// SIMATIC S7-200 project (STEP 7-Micro/WIN), CPU 226 REL 02.01

ORGANIZATION_BLOCK Main:OB1
TITLE=程序注释
BEGIN
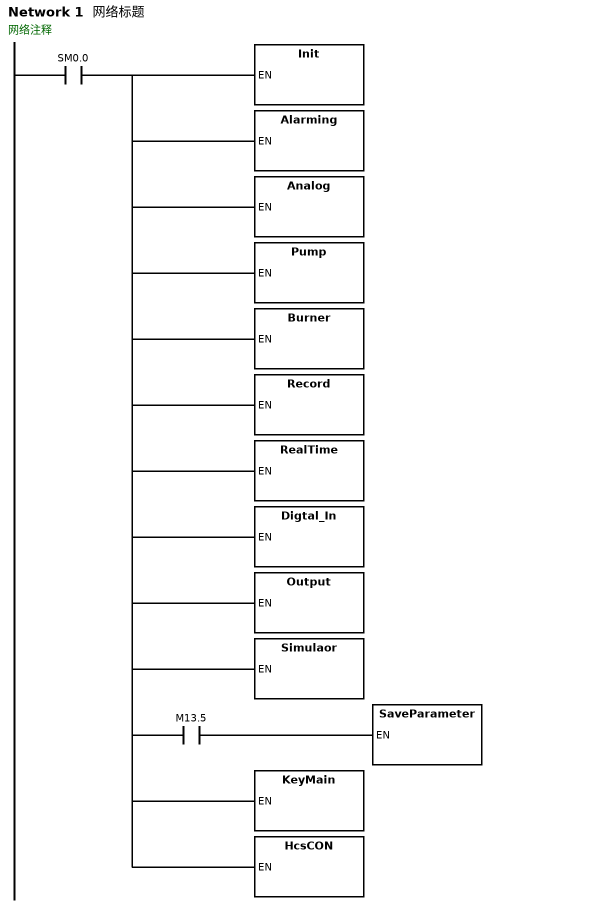
Network 1 // 网络标题
// 网络注释
LD     SM0.0
LPS
CALL   Init:SBR0
CALL   Alarming:SBR4
CALL   Analog:SBR1
CALL   Pump:SBR7
CALL   Burner:SBR14
CALL   Record:SBR11
CALL   RealTime:SBR19
CALL   Digtal_In:SBR17
CALL   Output:SBR24
CALL   Simulaor:SBR25
A      M13.5
CALL   SaveParameter:SBR26
LRD
CALL   KeyMain:SBR28
LPP
CALL   HcsCON:SBR32
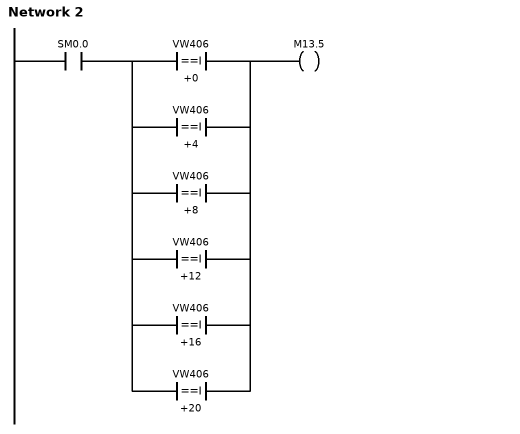
Network 2
LD     SM0.0
LDW=   VW406, +0
OW=    VW406, +4
OW=    VW406, +8
OW=    VW406, +12
OW=    VW406, +16
OW=    VW406, +20
ALD
=      M13.5
END_ORGANIZATION_BLOCK

SUBROUTINE_BLOCK Init:SBR0
TITLE=子程序注释
BEGIN
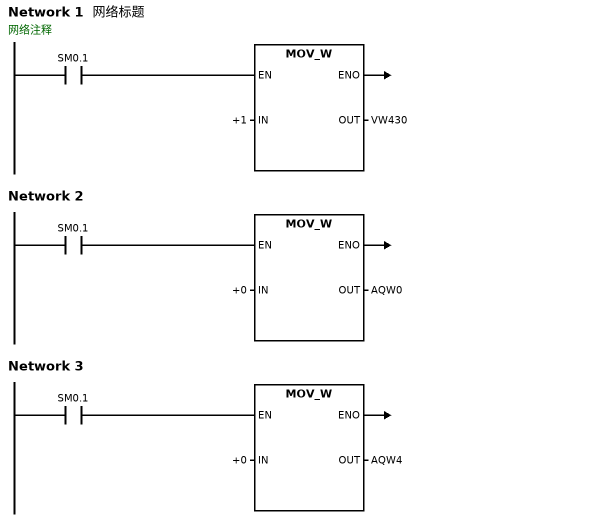
Network 1 // 网络标题
// 网络注释
LD     SM0.1
MOVW   +1, VW430
Network 2
LD     SM0.1
MOVW   +0, AQW0
Network 3
LD     SM0.1
MOVW   +0, AQW4
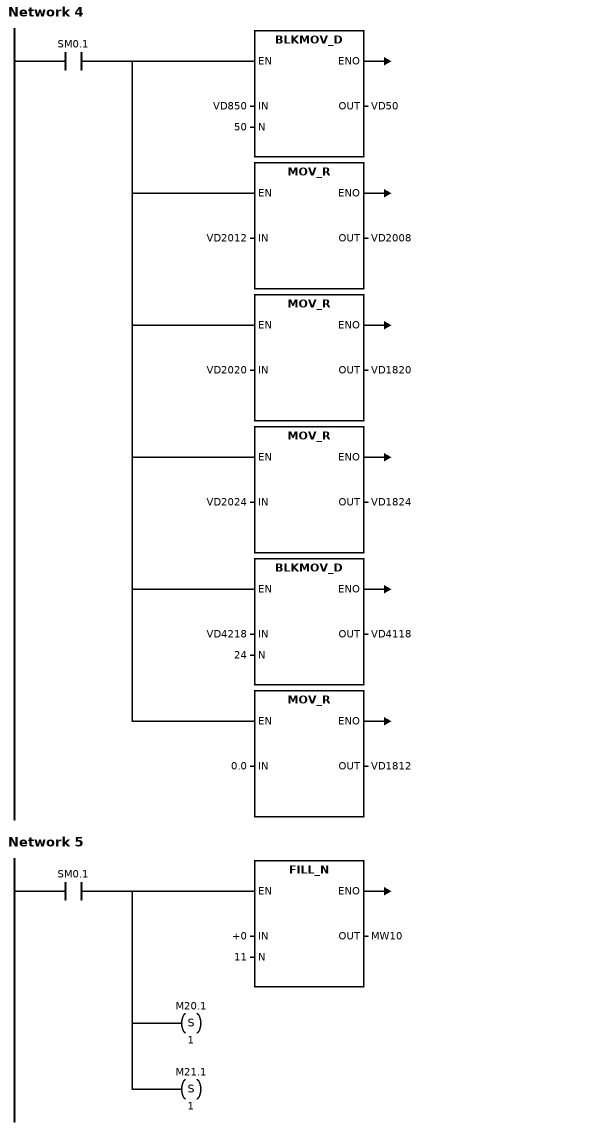
Network 4
LD     SM0.1
BMD    VD850, VD50, 50
MOVR   VD2012, VD2008
MOVR   VD2020, VD1820
MOVR   VD2024, VD1824
BMD    VD4218, VD4118, 24
MOVR   0.0, VD1812
Network 5
LD     SM0.1
FILL   +0, MW10, 11
S      M20.1, 1
S      M21.1, 1
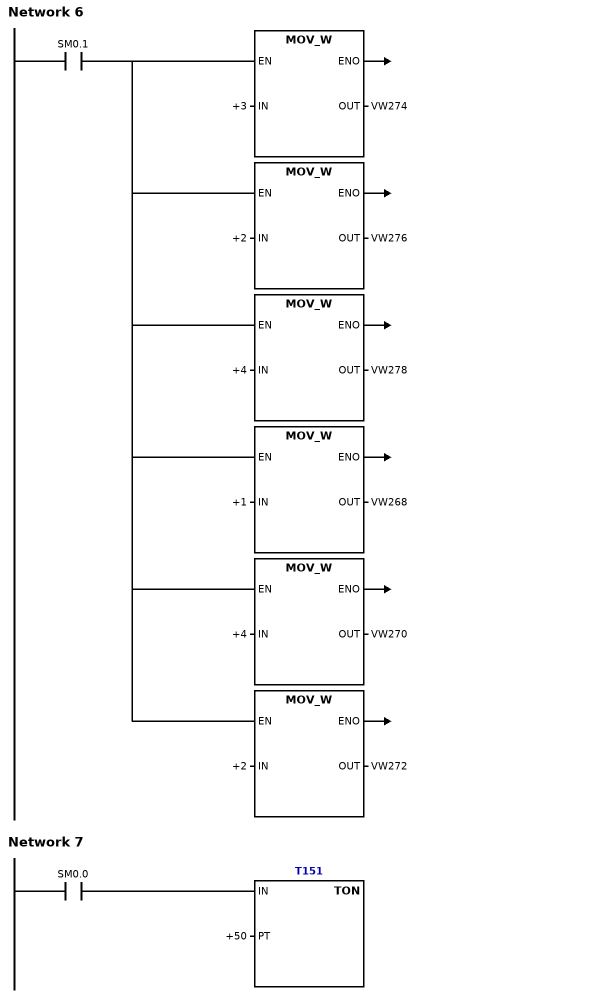
Network 6
LD     SM0.1
MOVW   +3, VW274
MOVW   +2, VW276
MOVW   +4, VW278
MOVW   +1, VW268
MOVW   +4, VW270
MOVW   +2, VW272
Network 7
LD     SM0.0
TON    T151, +50
END_SUBROUTINE_BLOCK

SUBROUTINE_BLOCK Analog:SBR1
TITLE=
BEGIN
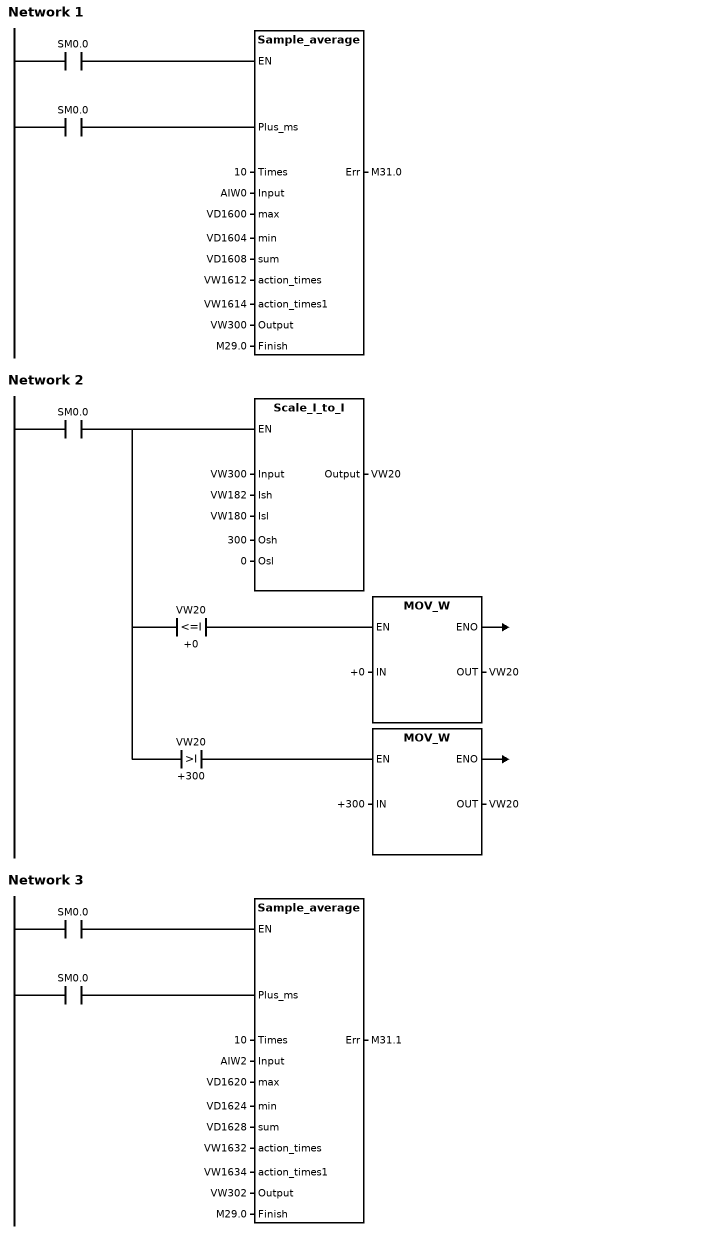
Network 1
LD     SM0.0
=      L60.0
LD     SM0.0
=      L63.7
LD     L60.0
CALL   Sample_average:SBR2, L63.7, 10, AIW0, VD1600, VD1604, VD1608, VW1612, VW1614, VW300, M29.0, M31.0
Network 2
LD     SM0.0
LPS
CALL   Scale_I_to_I:SBR3, VW300, VW182, VW180, 300, 0, VW20
AW<=   VW20, +0
MOVW   +0, VW20
LPP
AW>    VW20, +300
MOVW   +300, VW20
Network 3
LD     SM0.0
=      L60.0
LD     SM0.0
=      L63.7
LD     L60.0
CALL   Sample_average:SBR2, L63.7, 10, AIW2, VD1620, VD1624, VD1628, VW1632, VW1634, VW302, M29.0, M31.1
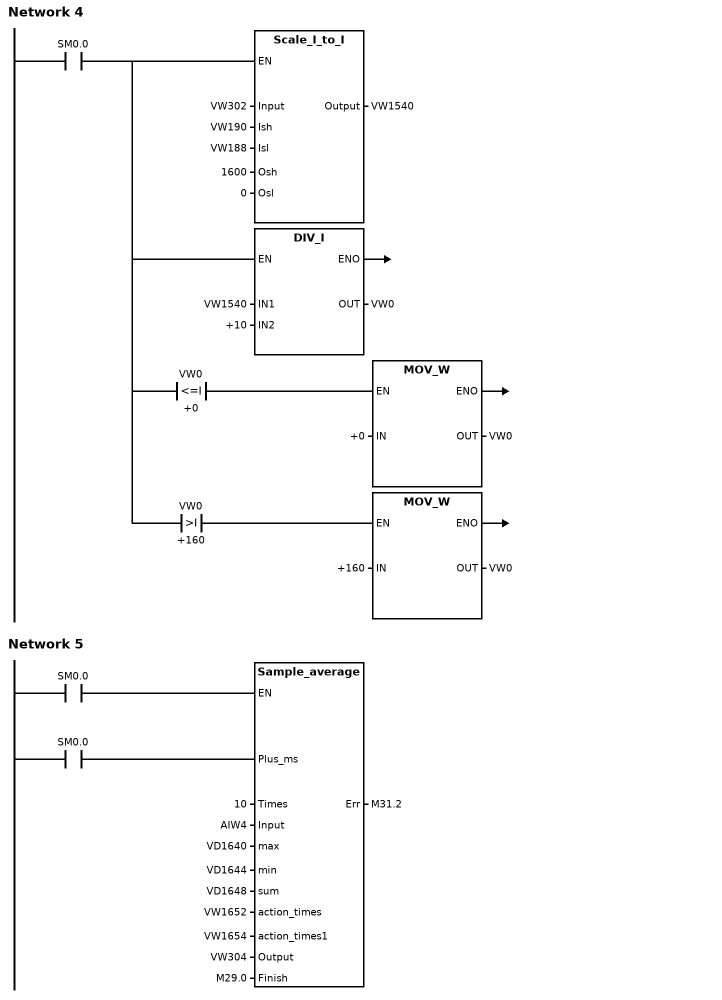
Network 4
LD     SM0.0
LPS
CALL   Scale_I_to_I:SBR3, VW302, VW190, VW188, 1600, 0, VW1540
MOVW   VW1540, VW0
/I     +10, VW0
AW<=   VW0, +0
MOVW   +0, VW0
LPP
AW>    VW0, +160
MOVW   +160, VW0
Network 5
LD     SM0.0
=      L60.0
LD     SM0.0
=      L63.7
LD     L60.0
CALL   Sample_average:SBR2, L63.7, 10, AIW4, VD1640, VD1644, VD1648, VW1652, VW1654, VW304, M29.0, M31.2
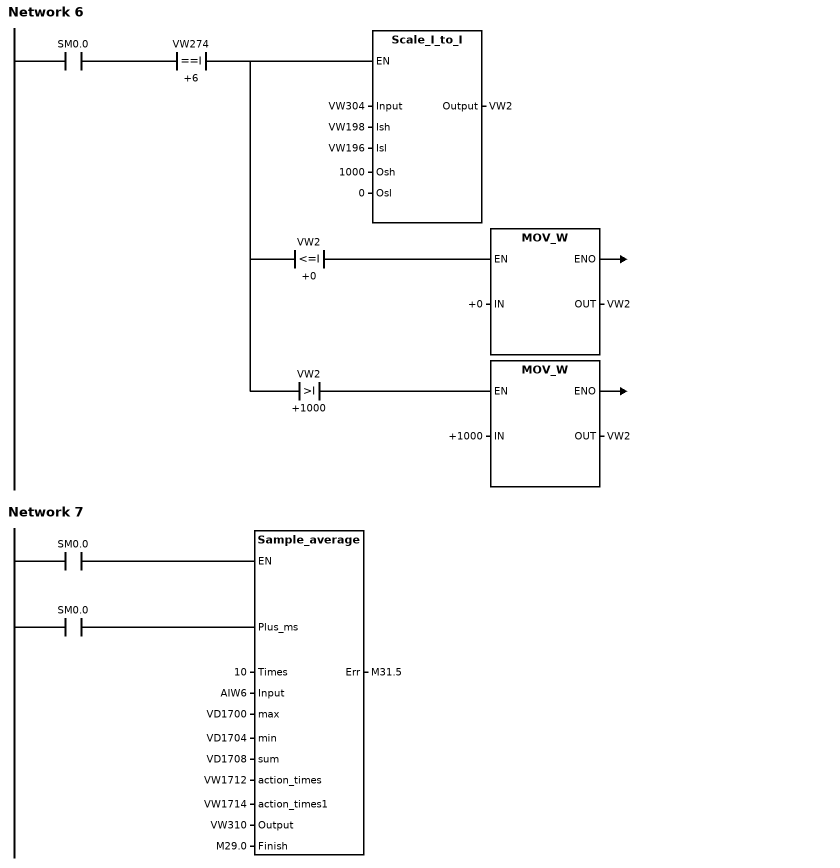
Network 6
LD     SM0.0
AW=    VW274, +6
LPS
CALL   Scale_I_to_I:SBR3, VW304, VW198, VW196, 1000, 0, VW2
AW<=   VW2, +0
MOVW   +0, VW2
LPP
AW>    VW2, +1000
MOVW   +1000, VW2
Network 7
LD     SM0.0
=      L60.0
LD     SM0.0
=      L63.7
LD     L60.0
CALL   Sample_average:SBR2, L63.7, 10, AIW6, VD1700, VD1704, VD1708, VW1712, VW1714, VW310, M29.0, M31.5
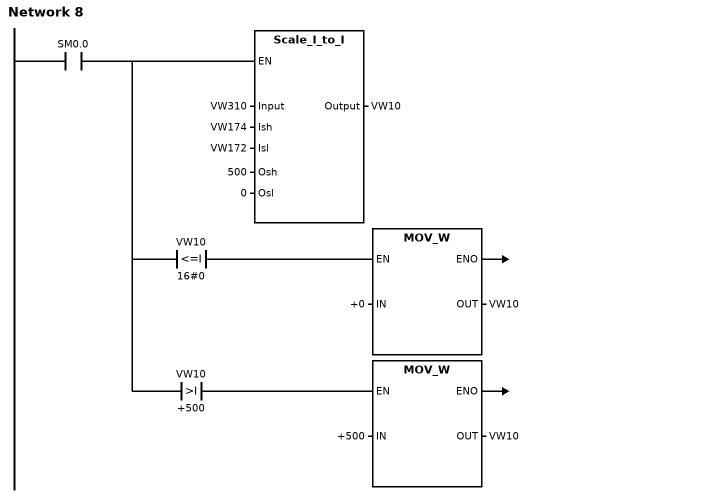
Network 8
LD     SM0.0
LPS
CALL   Scale_I_to_I:SBR3, VW310, VW174, VW172, 500, 0, VW10
AW<=   VW10, 16#0
MOVW   +0, VW10
LPP
AW>    VW10, +500
MOVW   +500, VW10
END_SUBROUTINE_BLOCK

SUBROUTINE_BLOCK Sample_average:SBR2
TITLE=
VAR_INPUT
Plus_ms:BOOL;	// L0.0 
Times:WORD;	// LW1 
Input:WORD;	// LW3 
END_VAR
VAR_IN_OUT
max:DWORD;	// LD5 
min:DWORD;	// LD9 
sum:DWORD;	// LD13 
action_times:WORD;	// LW17 
action_times1:WORD;	// LW19 
Output:WORD;	// LW21 
Finish:BOOL;	// L23.0 
END_VAR
VAR_OUTPUT
Err:BOOL;	// L23.1 
END_VAR
BEGIN
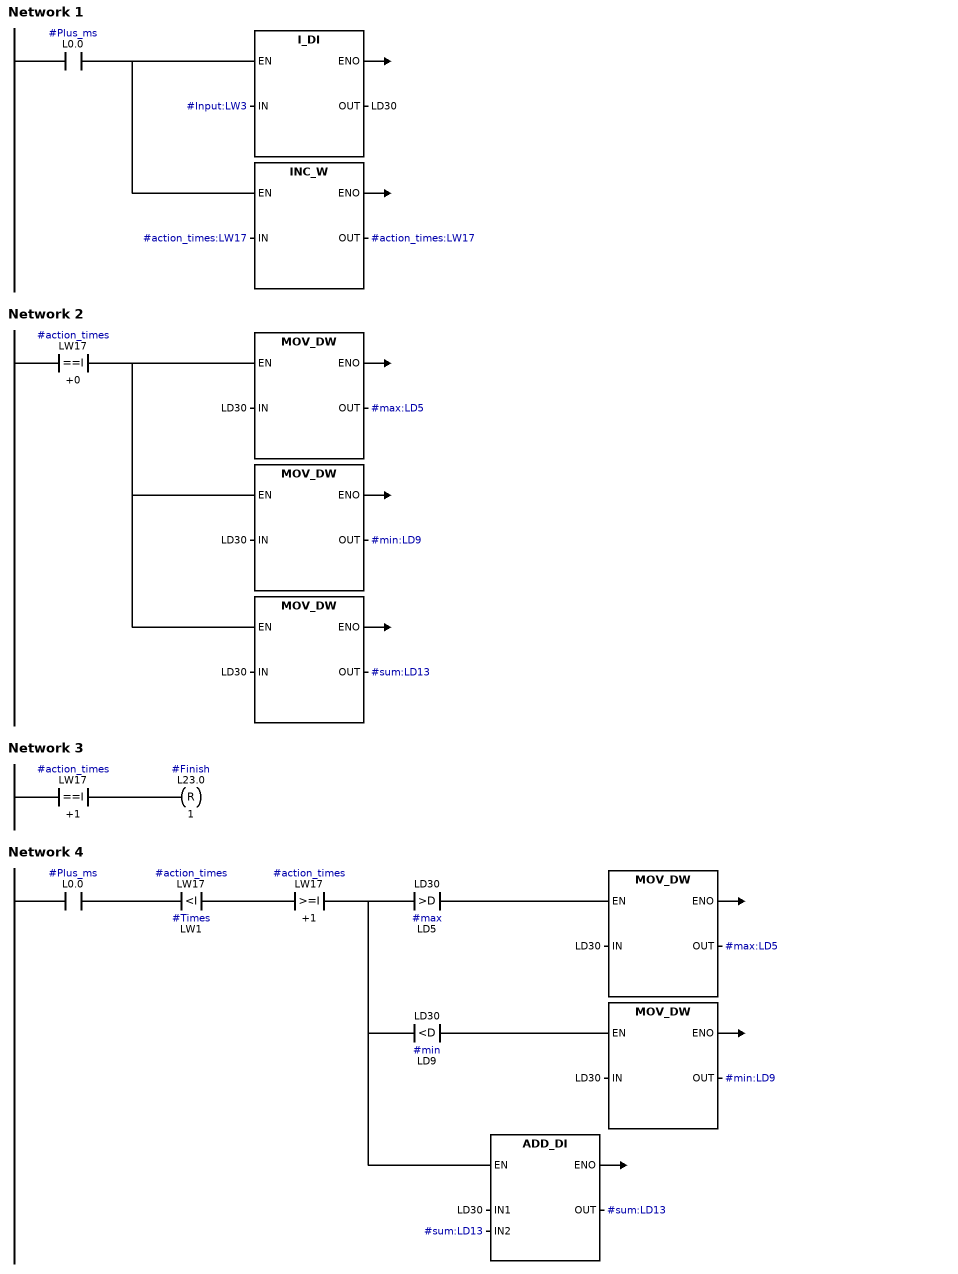
Network 1
LD     #Plus_ms:L0.0
ITD    #Input:LW3, LD30
INCW   #action_times:LW17
Network 2
LDW=   #action_times:LW17, +0
MOVD   LD30, #max:LD5
MOVD   LD30, #min:LD9
MOVD   LD30, #sum:LD13
Network 3
LDW=   #action_times:LW17, +1
R      #Finish:L23.0, 1
Network 4
LD     #Plus_ms:L0.0
AW<    #action_times:LW17, #Times:LW1
AW>=   #action_times:LW17, +1
LPS
AD>    LD30, #max:LD5
MOVD   LD30, #max:LD5
LRD
AD<    LD30, #min:LD9
MOVD   LD30, #min:LD9
LPP
+D     LD30, #sum:LD13
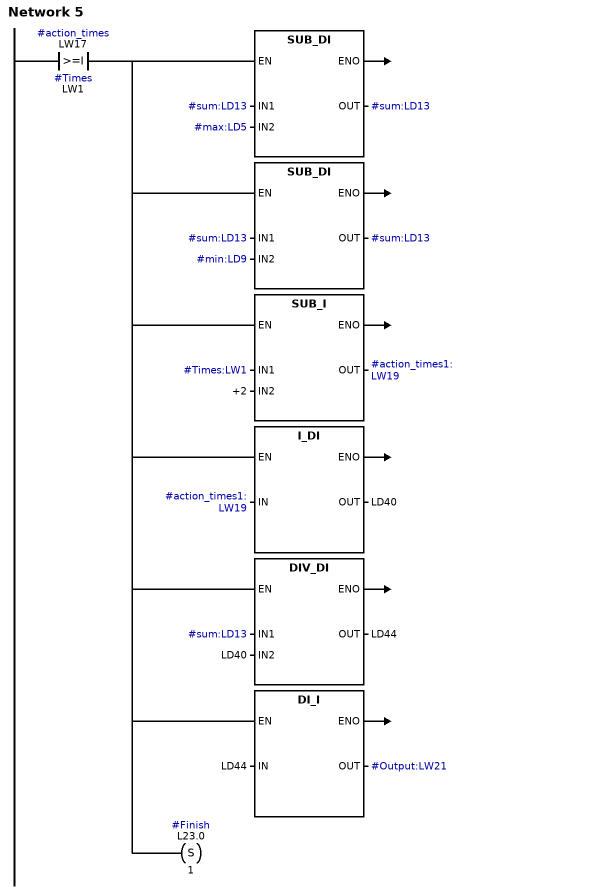
Network 5
LDW>=  #action_times:LW17, #Times:LW1
-D     #max:LD5, #sum:LD13
-D     #min:LD9, #sum:LD13
MOVW   #Times:LW1, #action_times1:LW19
-I     +2, #action_times1:LW19
ITD    #action_times1:LW19, LD40
MOVD   #sum:LD13, LD44
/D     LD40, LD44
DTI    LD44, #Output:LW21
S      #Finish:L23.0, 1
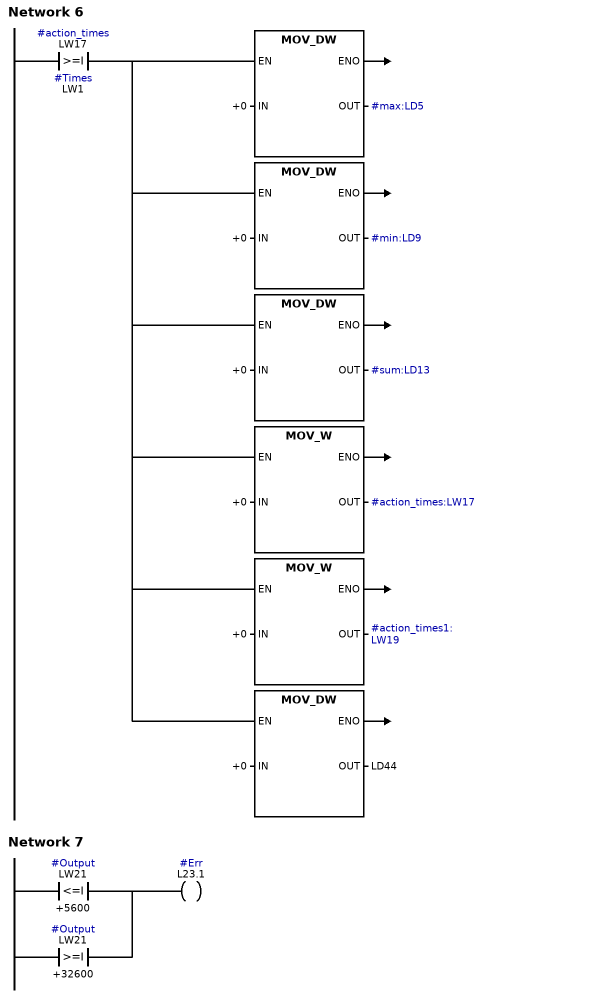
Network 6
LDW>=  #action_times:LW17, #Times:LW1
MOVD   +0, #max:LD5
MOVD   +0, #min:LD9
MOVD   +0, #sum:LD13
MOVW   +0, #action_times:LW17
MOVW   +0, #action_times1:LW19
MOVD   +0, LD44
Network 7
LDW<=  #Output:LW21, +5600
OW>=   #Output:LW21, +32600
=      #Err:L23.1
END_SUBROUTINE_BLOCK

// SBR3: protected block, not included

SUBROUTINE_BLOCK Alarming:SBR4
TITLE=
BEGIN
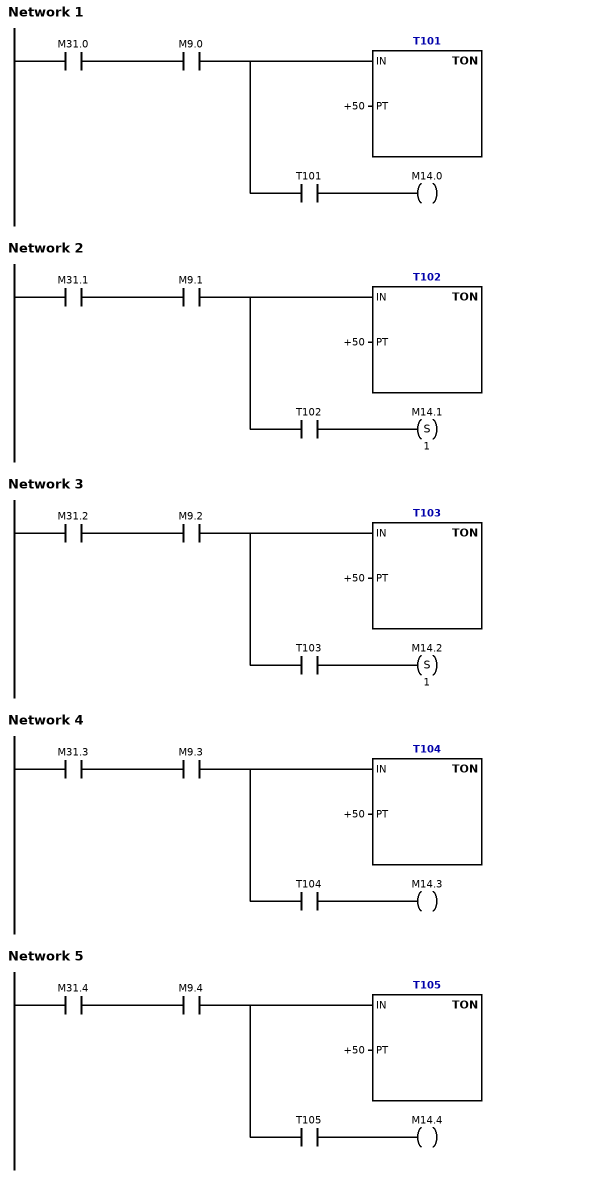
Network 1
LD     M31.0
A      M9.0
TON    T101, +50
A      T101
=      M14.0
Network 2
LD     M31.1
A      M9.1
TON    T102, +50
A      T102
S      M14.1, 1
Network 3
LD     M31.2
A      M9.2
TON    T103, +50
A      T103
S      M14.2, 1
Network 4
LD     M31.3
A      M9.3
TON    T104, +50
A      T104
=      M14.3
Network 5
LD     M31.4
A      M9.4
TON    T105, +50
A      T105
=      M14.4
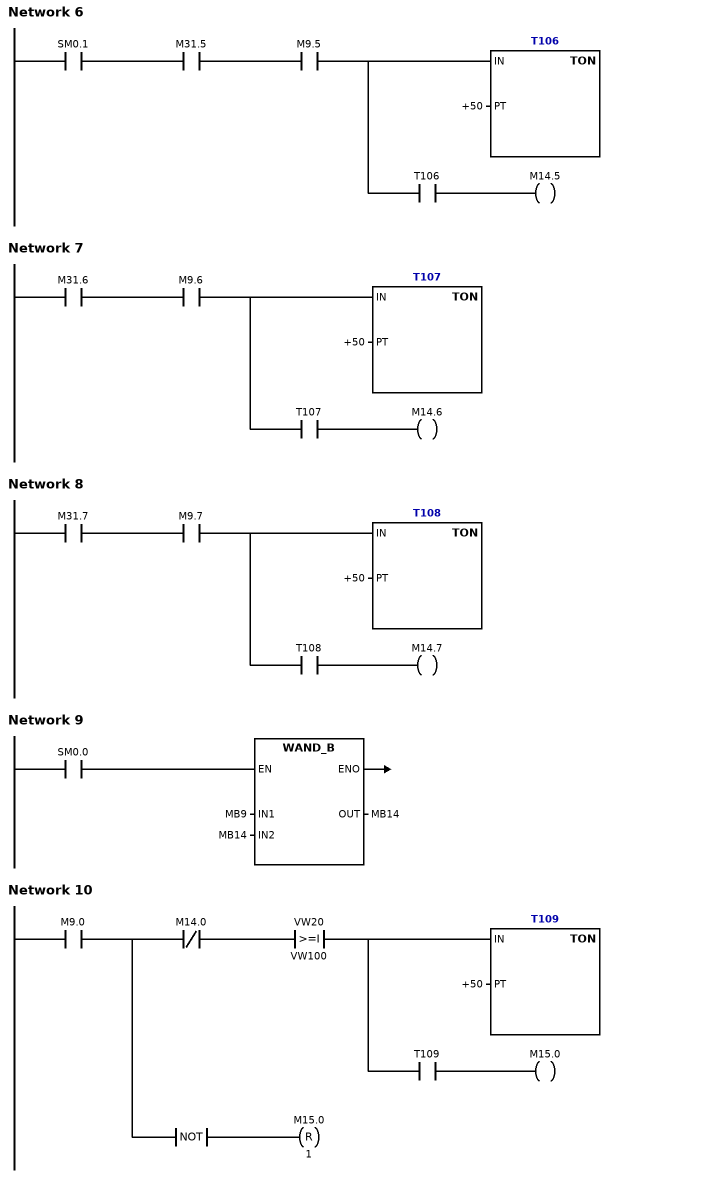
Network 6
LD     SM0.1
A      M31.5
A      M9.5
TON    T106, +50
A      T106
=      M14.5
Network 7
LD     M31.6
A      M9.6
TON    T107, +50
A      T107
=      M14.6
Network 8
LD     M31.7
A      M9.7
TON    T108, +50
A      T108
=      M14.7
Network 9
LD     SM0.0
ANDB   MB9, MB14
Network 10
LD     M9.0
LPS
AN     M14.0
AW>=   VW20, VW100
TON    T109, +50
A      T109
=      M15.0
LPP
NOT
R      M15.0, 1
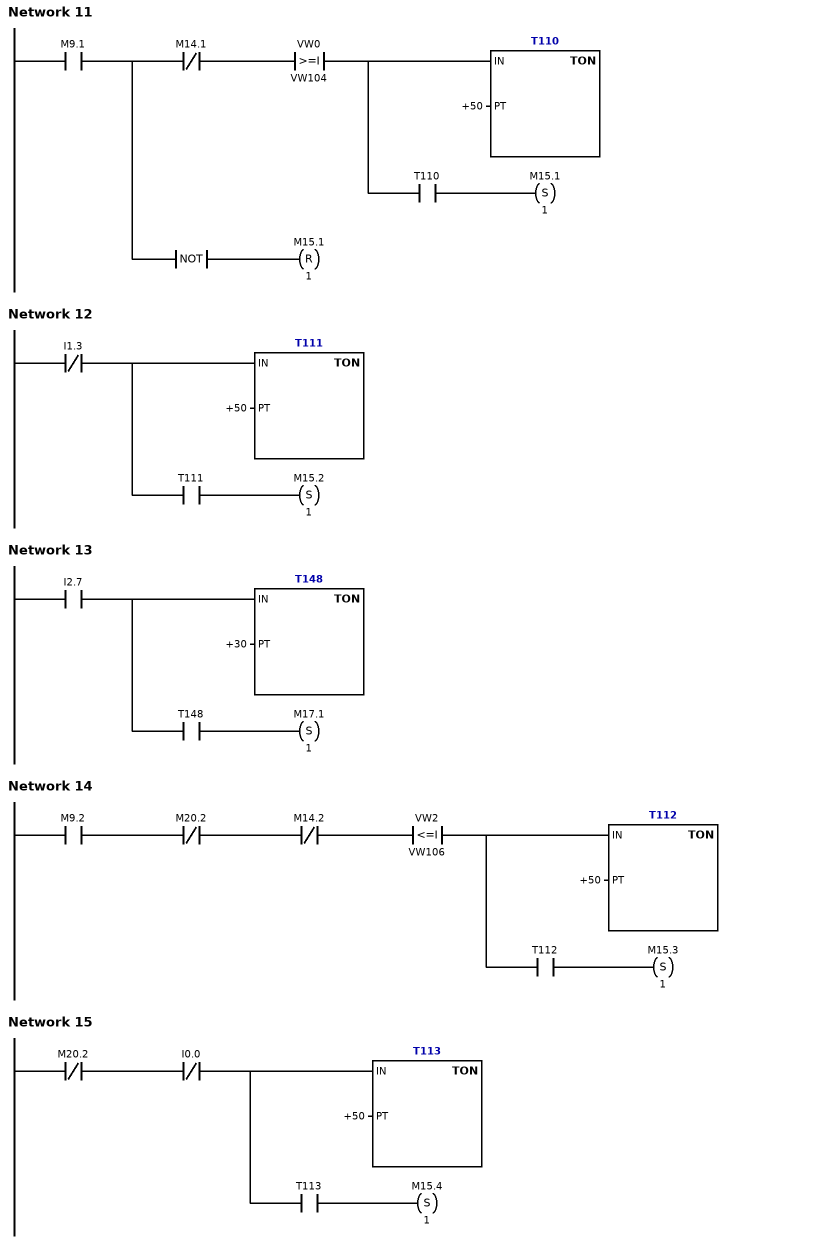
Network 11
LD     M9.1
LPS
AN     M14.1
AW>=   VW0, VW104
TON    T110, +50
A      T110
S      M15.1, 1
LPP
NOT
R      M15.1, 1
Network 12
LDN    I1.3
TON    T111, +50
A      T111
S      M15.2, 1
Network 13
LD     I2.7
TON    T148, +30
A      T148
S      M17.1, 1
Network 14
LD     M9.2
AN     M20.2
AN     M14.2
AW<=   VW2, VW106
TON    T112, +50
A      T112
S      M15.3, 1
Network 15
LDN    M20.2
AN     I0.0
TON    T113, +50
A      T113
S      M15.4, 1
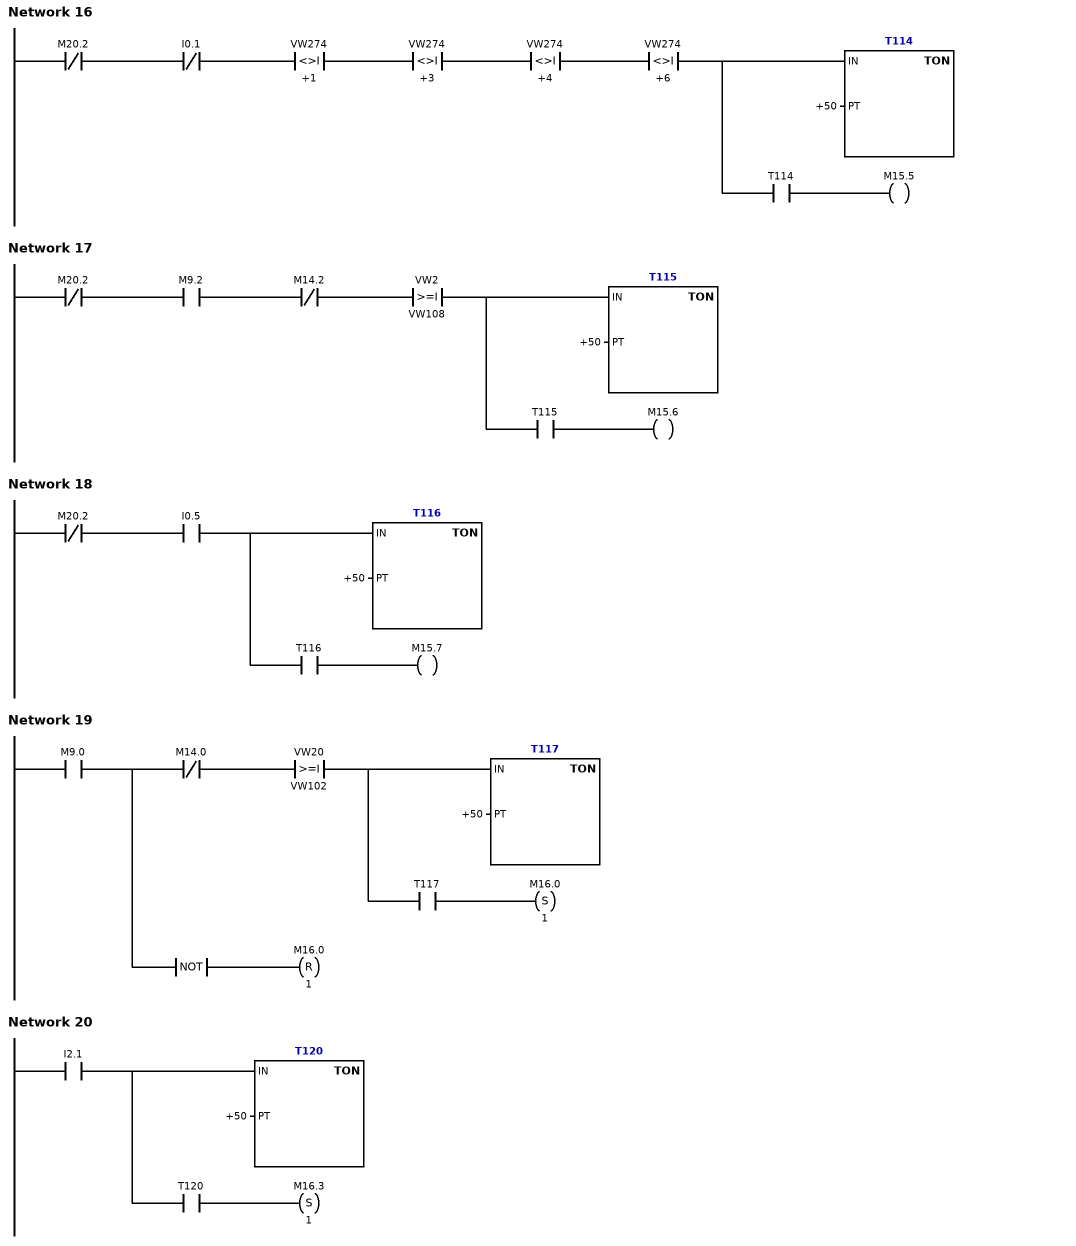
Network 16
LDN    M20.2
AN     I0.1
AW<>   VW274, +1
AW<>   VW274, +3
AW<>   VW274, +4
AW<>   VW274, +6
TON    T114, +50
A      T114
=      M15.5
Network 17
LDN    M20.2
A      M9.2
AN     M14.2
AW>=   VW2, VW108
TON    T115, +50
A      T115
=      M15.6
Network 18
LDN    M20.2
A      I0.5
TON    T116, +50
A      T116
=      M15.7
Network 19
LD     M9.0
LPS
AN     M14.0
AW>=   VW20, VW102
TON    T117, +50
A      T117
S      M16.0, 1
LPP
NOT
R      M16.0, 1
Network 20
LD     I2.1
TON    T120, +50
A      T120
S      M16.3, 1
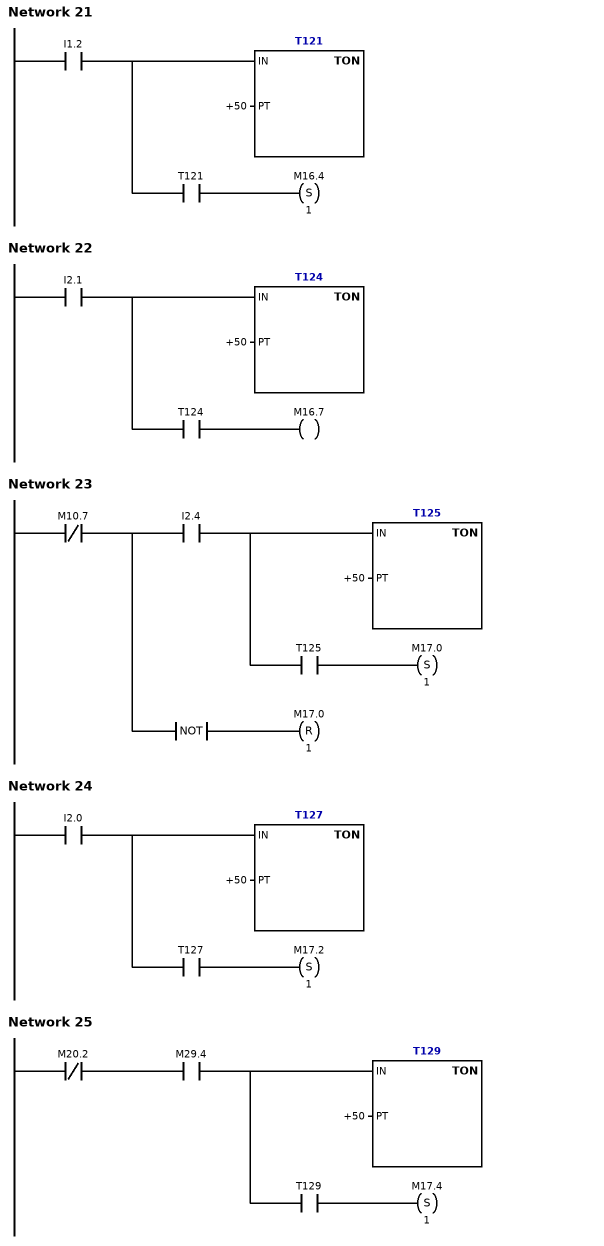
Network 21
LD     I1.2
TON    T121, +50
A      T121
S      M16.4, 1
Network 22
LD     I2.1
TON    T124, +50
A      T124
=      M16.7
Network 23
LDN    M10.7
LPS
A      I2.4
TON    T125, +50
A      T125
S      M17.0, 1
LPP
NOT
R      M17.0, 1
Network 24
LD     I2.0
TON    T127, +50
A      T127
S      M17.2, 1
Network 25
LDN    M20.2
A      M29.4
TON    T129, +50
A      T129
S      M17.4, 1
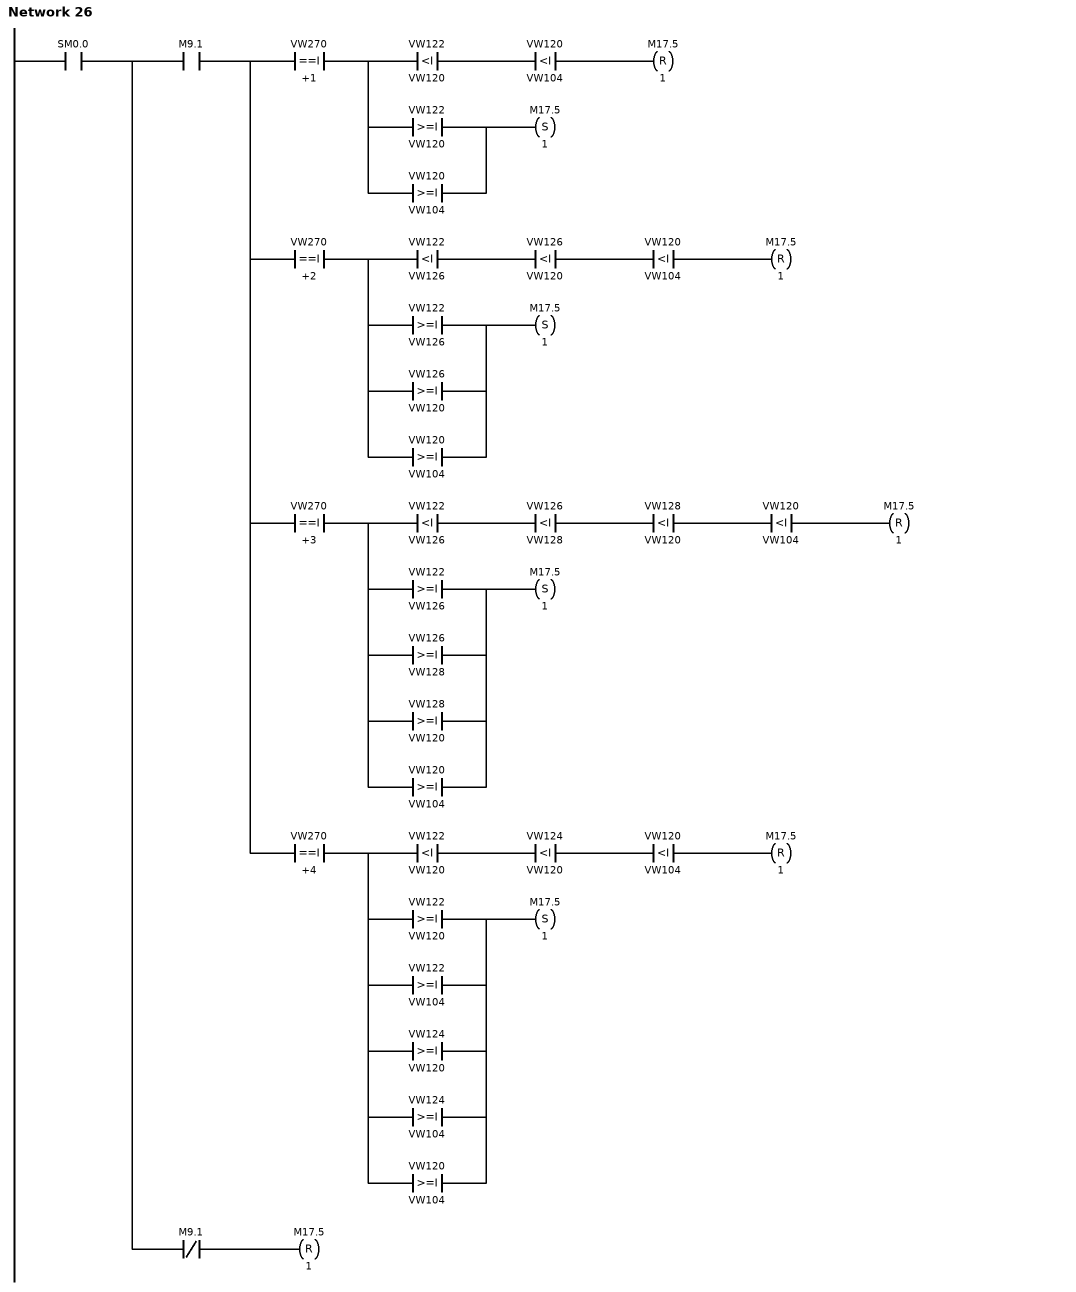
Network 26
LD     SM0.0
LPS
A      M9.1
LPS
AW=    VW270, +1
LPS
AW<    VW122, VW120
AW<    VW120, VW104
R      M17.5, 1
LPP
LDW>=  VW122, VW120
OW>=   VW120, VW104
ALD
S      M17.5, 1
LRD
AW=    VW270, +2
LPS
AW<    VW122, VW126
AW<    VW126, VW120
AW<    VW120, VW104
R      M17.5, 1
LPP
LDW>=  VW122, VW126
OW>=   VW126, VW120
OW>=   VW120, VW104
ALD
S      M17.5, 1
LRD
AW=    VW270, +3
LPS
AW<    VW122, VW126
AW<    VW126, VW128
AW<    VW128, VW120
AW<    VW120, VW104
R      M17.5, 1
LPP
LDW>=  VW122, VW126
OW>=   VW126, VW128
OW>=   VW128, VW120
OW>=   VW120, VW104
ALD
S      M17.5, 1
LPP
AW=    VW270, +4
LPS
AW<    VW122, VW120
AW<    VW124, VW120
AW<    VW120, VW104
R      M17.5, 1
LPP
LDW>=  VW122, VW120
OW>=   VW122, VW104
OW>=   VW124, VW120
OW>=   VW124, VW104
OW>=   VW120, VW104
ALD
S      M17.5, 1
LPP
AN     M9.1
R      M17.5, 1
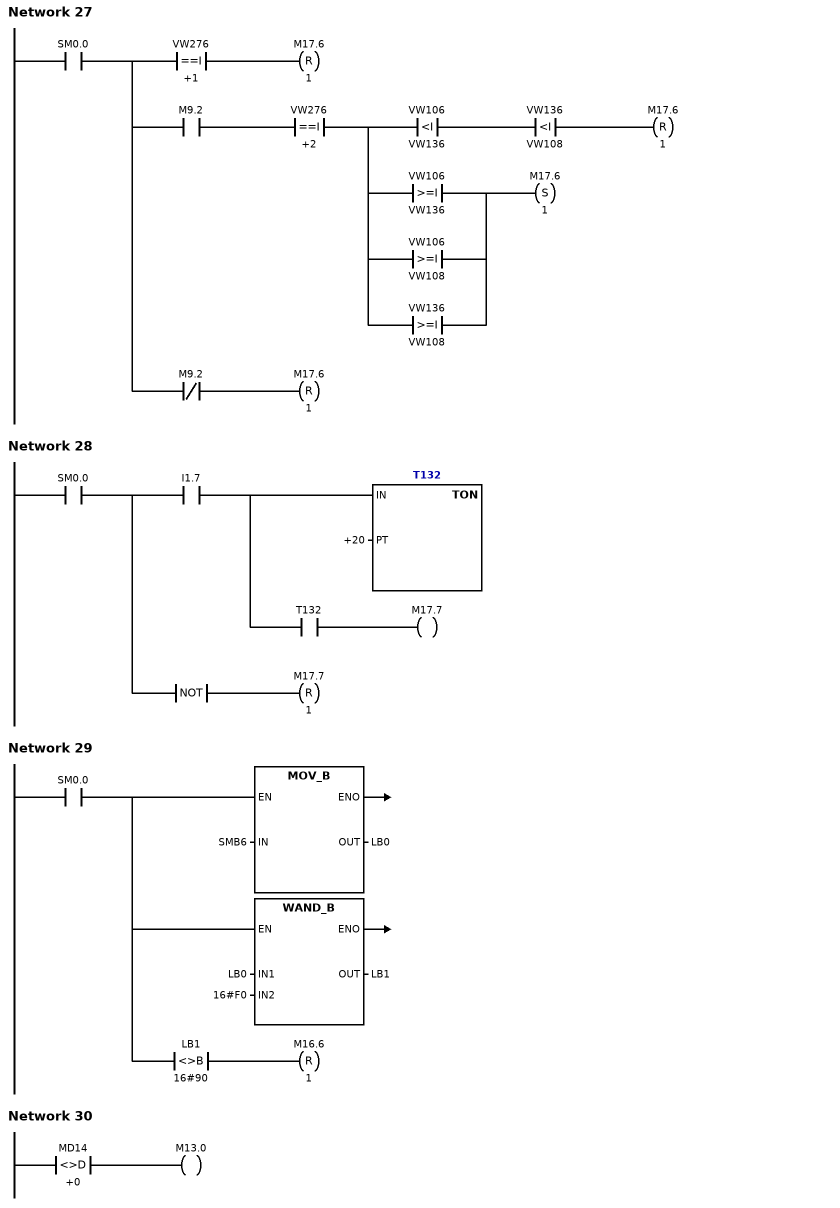
Network 27
LD     SM0.0
LPS
AW=    VW276, +1
R      M17.6, 1
LRD
A      M9.2
AW=    VW276, +2
LPS
AW<    VW106, VW136
AW<    VW136, VW108
R      M17.6, 1
LPP
LDW>=  VW106, VW136
OW>=   VW106, VW108
OW>=   VW136, VW108
ALD
S      M17.6, 1
LPP
AN     M9.2
R      M17.6, 1
Network 28
LD     SM0.0
LPS
A      I1.7
TON    T132, +20
A      T132
=      M17.7
LPP
NOT
R      M17.7, 1
Network 29
LD     SM0.0
MOVB   SMB6, LB0
MOVB   LB0, LB1
ANDB   16#F0, LB1
AB<>   LB1, 16#90
R      M16.6, 1
Network 30
LDD<>  MD14, +0
=      M13.0
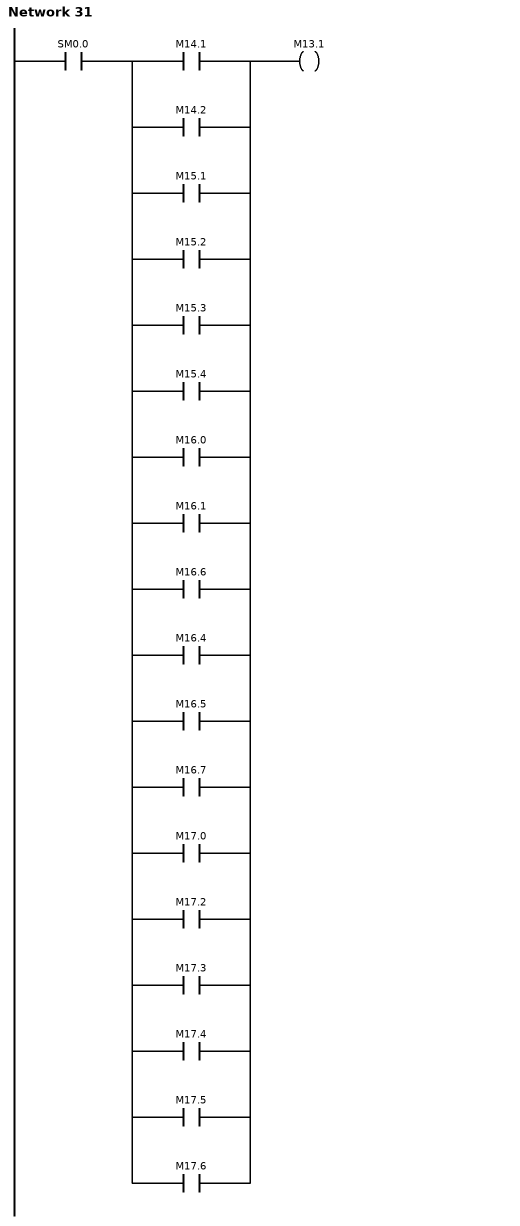
Network 31
LD     SM0.0
LD     M14.1
O      M14.2
O      M15.1
O      M15.2
O      M15.3
O      M15.4
O      M16.0
O      M16.1
O      M16.6
O      M16.4
O      M16.5
O      M16.7
O      M17.0
O      M17.2
O      M17.3
O      M17.4
O      M17.5
O      M17.6
ALD
=      M13.1
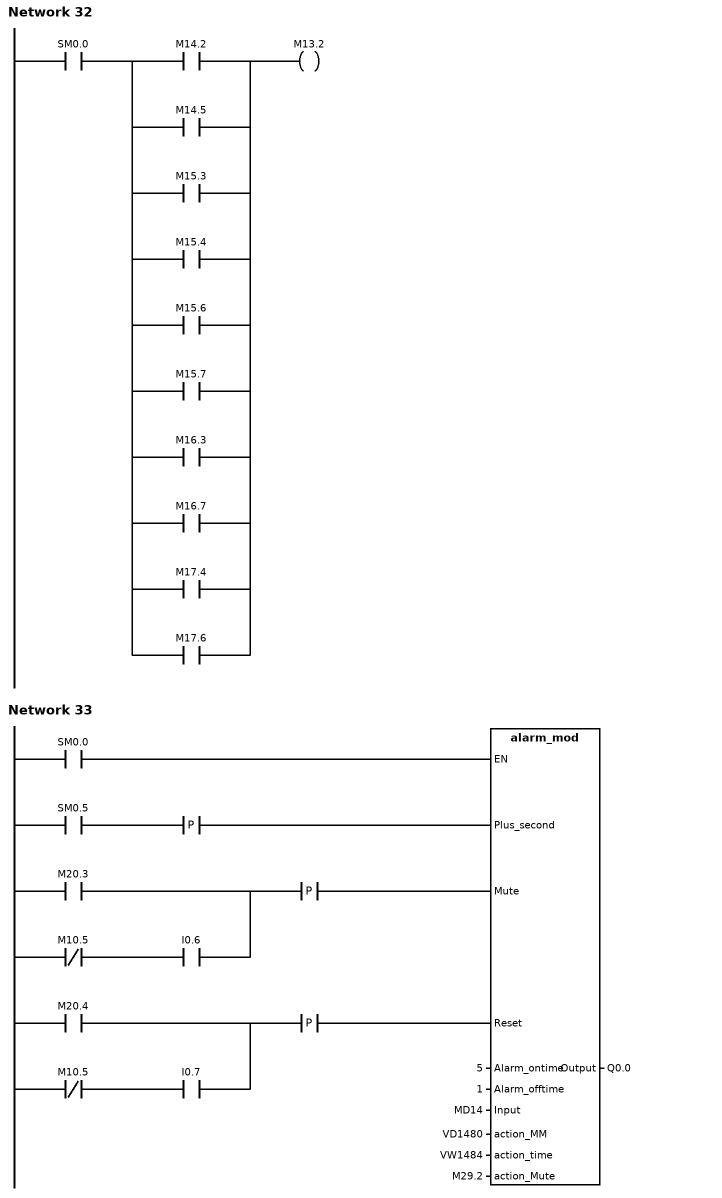
Network 32
LD     SM0.0
LD     M14.2
O      M14.5
O      M15.3
O      M15.4
O      M15.6
O      M15.7
O      M16.3
O      M16.7
O      M17.4
O      M17.6
ALD
=      M13.2
Network 33
LD     SM0.0
=      L60.0
LD     SM0.5
EU
=      L63.7
LD     M20.3
LDN    M10.5
A      I0.6
OLD
EU
=      L63.6
LD     M20.4
LDN    M10.5
A      I0.7
OLD
EU
=      L63.5
LD     L60.0
CALL   alarm_mod:SBR5, L63.7, L63.6, L63.5, 5, 1, MD14, VD1480, VW1484, M29.2, Q0.0
END_SUBROUTINE_BLOCK

// SBR5: protected block, not included

// SBR6: protected block, not included

SUBROUTINE_BLOCK Pump:SBR7
TITLE=
BEGIN
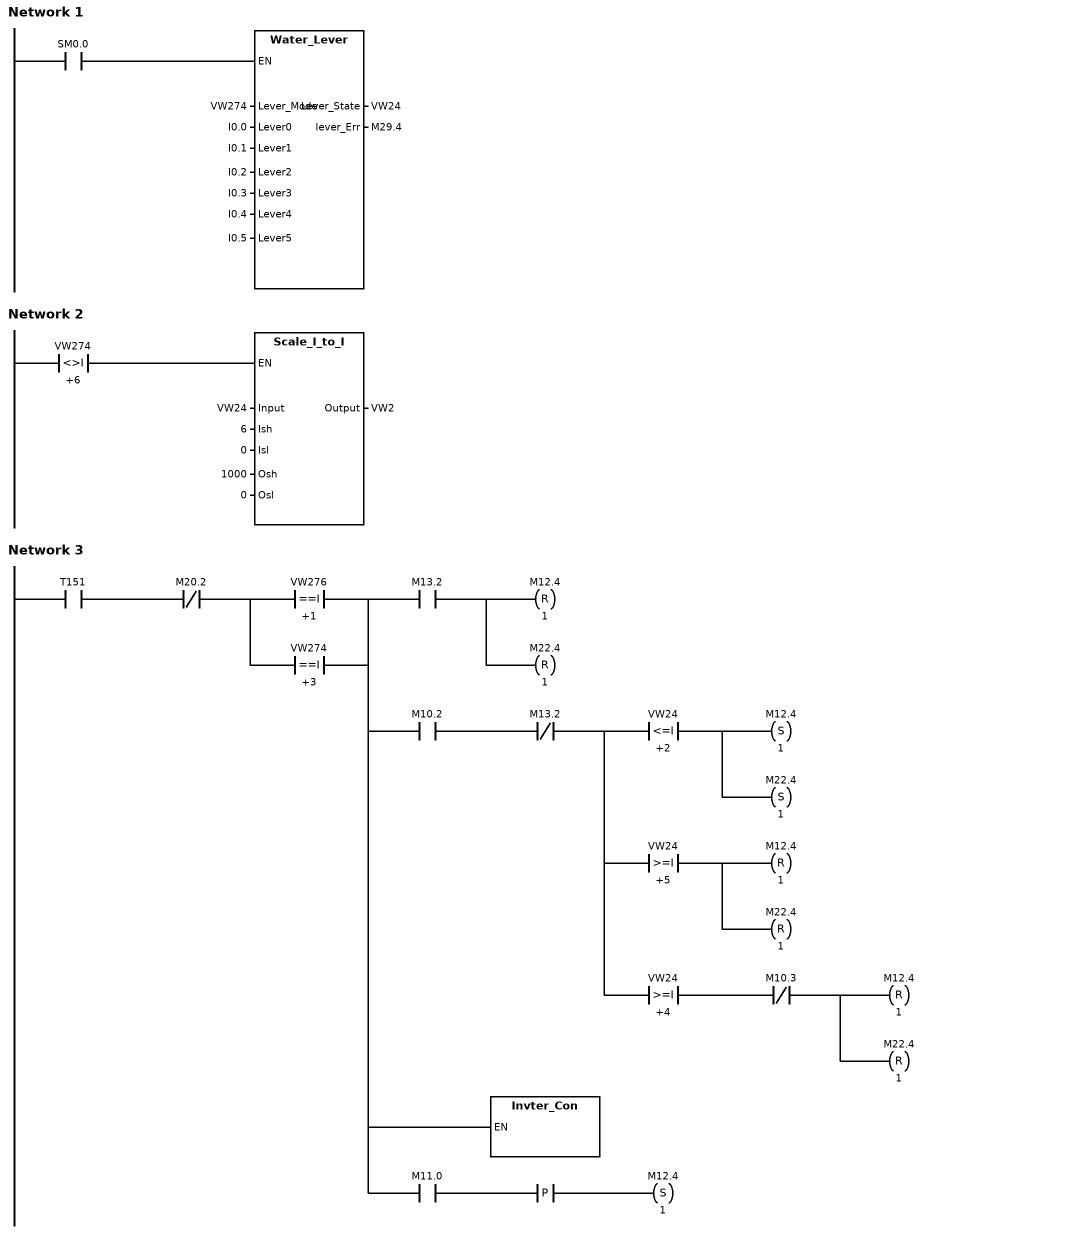
Network 1
LD     SM0.0
CALL   Water_Lever:SBR8, VW274, I0.0, I0.1, I0.2, I0.3, I0.4, I0.5, VW24, M29.4
Network 2
LDW<>  VW274, +6
CALL   Scale_I_to_I:SBR3, VW24, 6, 0, 1000, 0, VW2
Network 3
LD     T151
AN     M20.2
LDW=   VW276, +1
OW=    VW274, +3
ALD
LPS
A      M13.2
R      M12.4, 1
R      M22.4, 1
LRD
A      M10.2
AN     M13.2
LPS
AW<=   VW24, +2
S      M12.4, 1
S      M22.4, 1
LRD
AW>=   VW24, +5
R      M12.4, 1
R      M22.4, 1
LPP
AW>=   VW24, +4
AN     M10.3
R      M12.4, 1
R      M22.4, 1
LPP
CALL   Invter_Con:SBR15
A      M11.0
EU
S      M12.4, 1
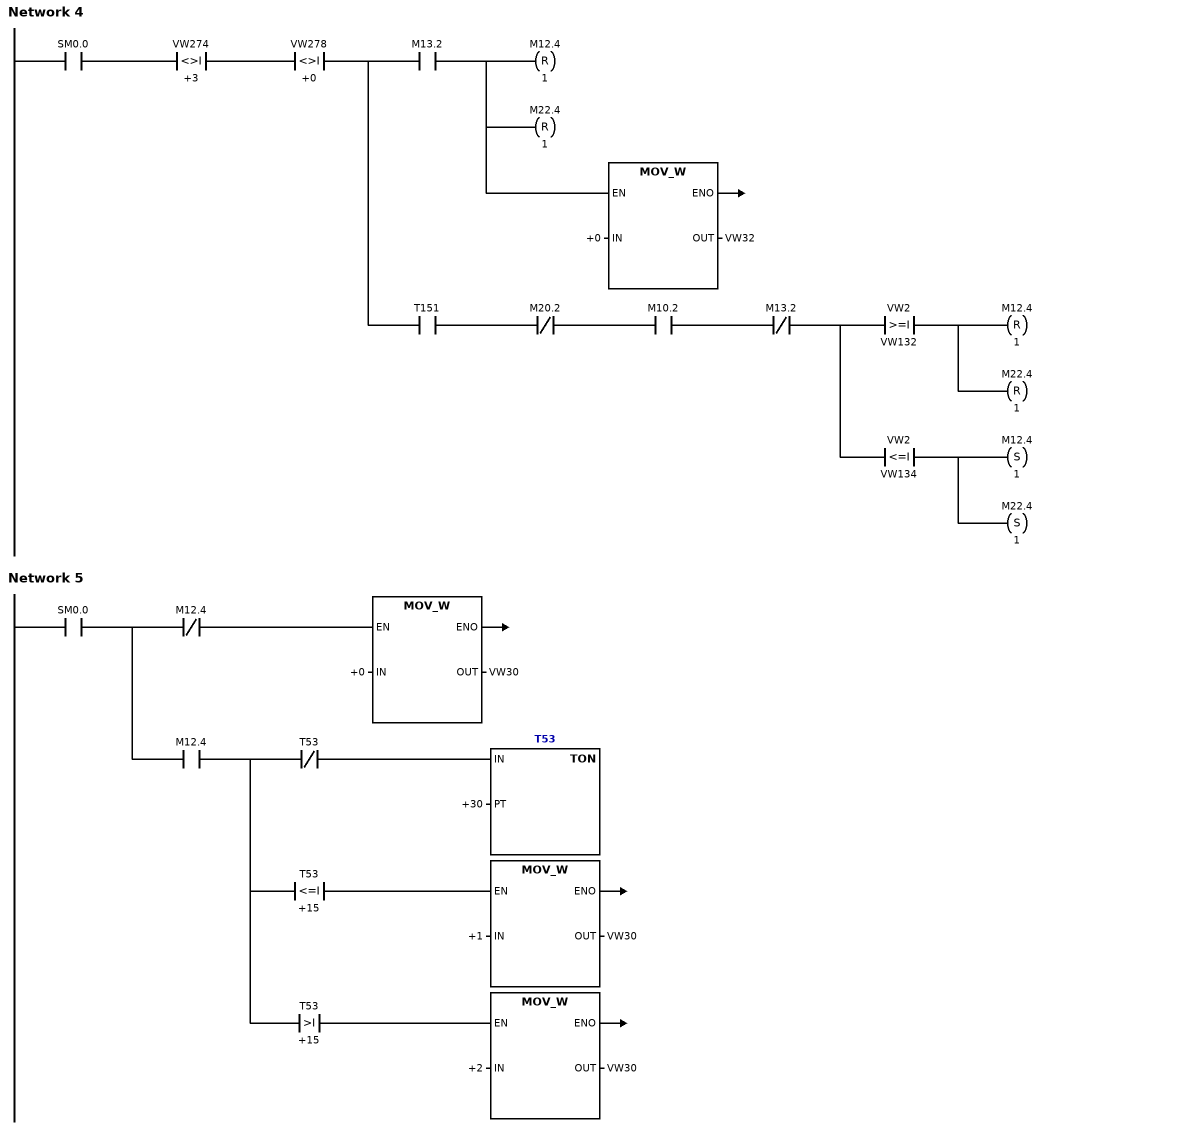
Network 4
LD     SM0.0
AW<>   VW274, +3
AW<>   VW278, +0
LPS
A      M13.2
R      M12.4, 1
R      M22.4, 1
MOVW   +0, VW32
LPP
A      T151
AN     M20.2
A      M10.2
AN     M13.2
LPS
AW>=   VW2, VW132
R      M12.4, 1
R      M22.4, 1
LPP
AW<=   VW2, VW134
S      M12.4, 1
S      M22.4, 1
Network 5
LD     SM0.0
LPS
AN     M12.4
MOVW   +0, VW30
LPP
A      M12.4
LPS
AN     T53
TON    T53, +30
LRD
AW<=   T53, +15
MOVW   +1, VW30
LPP
AW>    T53, +15
MOVW   +2, VW30
END_SUBROUTINE_BLOCK

// SBR8: protected block, not included

// SBR9: protected block, not included

SUBROUTINE_BLOCK Record:SBR11
TITLE=
BEGIN
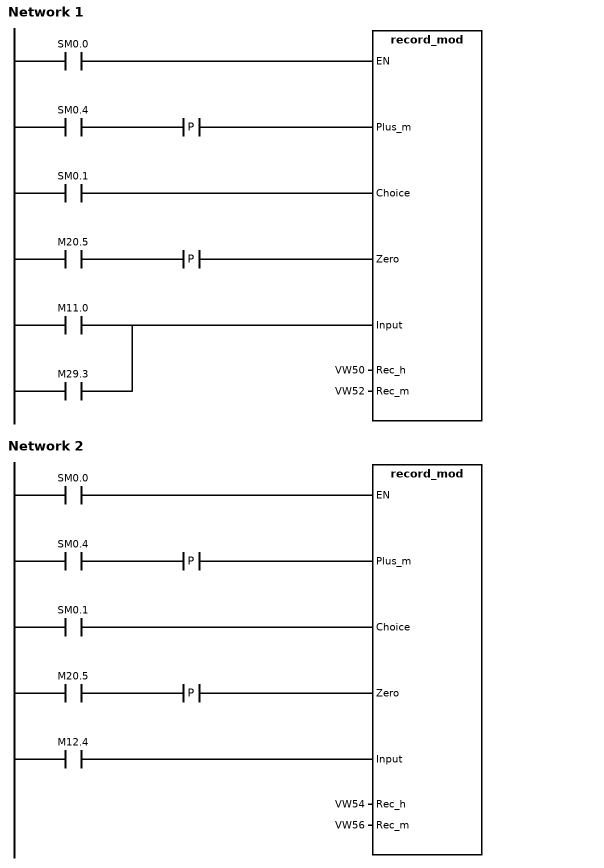
Network 1
LD     SM0.0
=      L60.0
LD     SM0.4
EU
=      L63.7
LD     SM0.1
=      L63.6
LD     M20.5
EU
=      L63.5
LD     M11.0
O      M29.3
=      L63.4
LD     L60.0
CALL   record_mod:SBR13, L63.7, L63.6, L63.5, L63.4, VW50, VW52
Network 2
LD     SM0.0
=      L60.0
LD     SM0.4
EU
=      L63.7
LD     SM0.1
=      L63.6
LD     M20.5
EU
=      L63.5
LD     M12.4
=      L63.4
LD     L60.0
CALL   record_mod:SBR13, L63.7, L63.6, L63.5, L63.4, VW54, VW56
